FUNCTION CheckDivSInt : SINT
VAR_INPUT
	divisor			 	: SINT;
END_VAR
VAR
END_VAR

IF divisor = 0 THEN
	CheckSIntZeroDiv_ErrCnt := CheckSIntZeroDiv_ErrCnt + 1;
	CheckDivSInt := 1;
ELSE
	CheckDivSInt := divisor;
END_IF

END_FUNCTION

(* stored: Version 1.1.0.1, ProductVersion 3.1.4024.9
   POU CheckDivSInt: Id {e7df892b-aa57-4a29-867e-0165a404fdfa}, SpecialFunc CheckDivInt32 *)
